(* CoDeSys 2.3 export: DEVICESTATUS.EXP *)

(* Data type in ENUM *)
TYPE DeviceStatus : (null:=0, alarm, stopped, started);
END_TYPE
